(* IEC 61131-3 sources: ToolBox/src/Ar/ToolBox, 6 files *)

(* ---- ToolBox.typ ---- *)
(*
 * File: ToolBox.typ
 * Copyright (c) 2023 Loupe
 * https://loupe.team
 *
 * This file is part of ToolBox, licensed under the MIT License.
 *
 *)

TYPE
	Process_Timer_Internal : 	STRUCT
		Timer : TON;
		NumberCounted : UDINT;
		StartCount : UDINT;
		CurrentCount : UDINT;
		CountTime : TIME;
		FilteredTime : TIME;
	END_STRUCT;
	TON_w_Pause_Internal : 	STRUCT
		PT : TIME;
		TimeLeft : TIME;
		TimerPaused : BOOL;
		ExecuteOnce : BOOL;
		TON_ : TON;
		TempET : TIME;
		Reset : BOOL;
	END_STRUCT;
END_TYPE

(* ---- WithinPercent.st ---- *)
(*
 * File: WithinPercent.st
 * Copyright (c) 2023 Loupe
 * https://loupe.team
 *
 * This file is part of ToolBox, licensed under the MIT License.
 *
 *)

(* simplify IF statements: if value is within a percentage window *)
FUNCTION WithinPercent
	IF SetValue <> 0 THEN
		WithinPercent := (ABS(SetValue - InputValue)/ABS(SetValue)) <= (PercentWindow/100.0);
	ELSE
		WithinPercent := InputValue = SetValue;
	END_IF;
END_FUNCTION

(* ---- ProcessTimer.st ---- *)
(*
 * File: ProcessTimer.st
 * Copyright (c) 2023 Loupe
 * https://loupe.team
 *
 * This file is part of ToolBox, licensed under the MIT License.
 *
 *)

(*  *)
FUNCTION_BLOCK ProcessTimer

	IF Reset THEN

		internal.Timer.IN:=0;
		internal.StartCount:=Count+1;
		internal.CurrentCount:=Count;
		internal.NumberCounted:=0;
		internal.CountTime:=0;
		internal.FilteredTime:=0;

	ELSIF Enable THEN

		IF internal.CurrentCount > Count THEN
			internal.CurrentCount:=Count;
			internal.StartCount:=Count+1;
		END_IF

		IF internal.StartCount < Count THEN

			internal.StartCount:=Count;
			internal.NumberCounted:=internal.NumberCounted+1;
			internal.CountTime:=internal.Timer.ET+internal.CountTime;

			IF internal.FilteredTime = 0 THEN

				internal.FilteredTime:= internal.Timer.ET;

			ELSE

				internal.FilteredTime:= (internal.FilteredTime*9+internal.Timer.ET)/10;

			END_IF

			internal.Timer.IN:=0;
			internal.Timer();
			internal.Timer.IN:=1;

		ELSIF internal.StartCount = Count THEN

			internal.Timer.IN:=1;

		END_IF

	ELSE

		internal.Timer.IN:=0;
		internal.StartCount:=Count+1;
		internal.CurrentCount:=Count;
	END_IF

	internal.Timer.PT:=1000000000;
	internal.Timer();

	FilteredTime:=internal.FilteredTime;

	IF internal.NumberCounted > 1 THEN
		AverageTime:=internal.CountTime/UDINT_TO_DINT(internal.NumberCounted);
	ELSE
		AverageTime:=0;
	END_IF

END_FUNCTION_BLOCK

(* ---- TON_Pause.st ---- *)
(*
 * File: TON_Pause.st
 * Copyright (c) 2023 Loupe
 * https://loupe.team
 *
 * This file is part of ToolBox, licensed under the MIT License.
 *
 *)

(* TON functionality with pausing and an output percentage *)
FUNCTION_BLOCK TON_Pause
	IF(IN) THEN
		IF (Internal.Reset) THEN
			Internal.Reset := 0;
			PercentCompleted := 0;
			Internal.TempET := 0;
		END_IF;

		IF(NOT Internal.ExecuteOnce) THEN
			Internal.PT :=	PT;
			Internal.TON_.PT := PT;
			Internal.TON_.IN := 1;
			Internal.ExecuteOnce := 1;
		END_IF;

		IF(Pause AND NOT Internal.TimerPaused)THEN
			IF (Q = 0)THEN
				Internal.TimeLeft :=    (Internal.TON_.PT - Internal.TON_.ET);
			ELSE
				Internal.TimeLeft := 0;
			END_IF;
			Internal.TempET := Internal.TempET + Internal.TON_.ET;
			Internal.TON_.IN := 0;
			Internal.TimerPaused := 1;
		END_IF;//end OF IF Pause

		Internal.TON_();

		IF ((Internal.TON_.Q = 0) AND (Internal.TON_.IN = 1))THEN
			ET := Internal.TempET + Internal.TON_.ET;
		END_IF;
		IF(NOT Pause AND Internal.TimerPaused)THEN
			Internal.TimerPaused := 0;
			Internal.TON_.PT := Internal.TimeLeft;
			Internal.TON_.IN := 1;
		END_IF;

		IF(Internal.TON_.Q)THEN
			Q := 1;
			Internal.TimeLeft := 0;
			Internal.TON_.IN := 0;
		END_IF;
		IF Q THEN
			TimeLeftRunning := 	0;
			PercentCompleted := 100;
			ET := Internal.PT;
		ELSE
			TimeLeftRunning := 	Internal.PT - ET;
			IF (Internal.PT <> 0)THEN
				PercentCompleted := ((TIME_TO_REAL(ET) * 100.0) / (TIME_TO_REAL(Internal.PT) * 100.0)) * 100.0;
			END_IF;
		END_IF;

	//End IF enabled
	ELSE
		Internal.Reset :=				1;
		Internal.PT :=	0;
		Internal.ExecuteOnce := 0;
		Internal.TimeLeft := 0;
		TimeLeftRunning := 0;
		Q := 0;
		Pause := 0;
		Internal.TON_.IN := 0;
		Internal.TimeLeft := 0;
		Internal.TimerPaused := 0;
		PercentCompleted := 0;
		ET :=	0;
		//FUB call to reset clock
		Internal.TON_();
	END_IF

END_FUNCTION_BLOCK

(* ---- ToolBox.fun ---- *)
(*
 * File: ToolBox.fun
 * Copyright (c) 2023 Loupe
 * https://loupe.team
 *
 * This file is part of ToolBox, licensed under the MIT License.
 *
 *)

FUNCTION_BLOCK ProcessTimer
	VAR_INPUT
		Enable : BOOL;
		Reset : BOOL;
		Count : UDINT;
	END_VAR
	VAR_OUTPUT
		AverageTime : TIME;
		FilteredTime : TIME;
	END_VAR
	VAR
		internal : Process_Timer_Internal;
	END_VAR
END_FUNCTION_BLOCK

FUNCTION_BLOCK TON_Pause (*TON functionality with pausing and an output percentage*) (*$GROUP=User,$CAT=User,$GROUPICON=LD_TimerCounter.png,$CATICON=User.png*)
	VAR_INPUT
		IN : BOOL;
		Pause : BOOL;
		PT : TIME;
	END_VAR
	VAR_OUTPUT
		Q : BOOL;
		ET : TIME;
		PercentCompleted : REAL;
		TimeLeftRunning : TIME;
	END_VAR
	VAR
		Internal : TON_w_Pause_Internal;
	END_VAR
END_FUNCTION_BLOCK

FUNCTION WithinPercent : BOOL (*simplify IF statement if value is within a percentage window*) (*$GROUP=User,$CAT=User,$GROUPICON=User.png,$CATICON=User.png*)
	VAR_INPUT
		InputValue : REAL; (*Value check*)
		SetValue : REAL; (*value to come close to*)
		PercentWindow : REAL; (*percentage window of SetInput that Input needs to be within [%]*)
	END_VAR
END_FUNCTION

(* ---- ToolBox.var ---- *)
(*
 * File: ToolBox.var
 * Copyright (c) 2023 Loupe
 * https://loupe.team
 *
 * This file is part of ToolBox, licensed under the MIT License.
 *
 *)

VAR CONSTANT

END_VAR
